            CASE is_COOLING_LEFT OF
                UPMRacing_14E_StateMachine_IN_COOLING_OFF_LEFT: 
                    (* During 'COOLING_OFF_LEFT': '<S1>:602' *)
                    (* '<S1>:603:1' sf_internal_predicateOutput = Cooling_Enable == true; *)

                    IF Cooling_Enable THEN 
                        (* Transition: '<S1>:603' *)
                        (* Exit 'COOLING_OFF_LEFT': '<S1>:602' *)
                        (* '<S1>:602:4' Cooling_Pumps_On = false; *)
                        Cooling_Pumps_On := FALSE;
                        is_COOLING_LEFT := UPMRacing_14E_StateMachine_IN_FAN_OFF;
                        (* Entry 'FAN_OFF': '<S1>:546' *)
                    END_IF;

                UPMRacing_14E_StateMachine_IN_FAN_OFF: 
                    (* During 'FAN_OFF': '<S1>:546' *)
                    (* '<S1>:548:1' sf_internal_predicateOutput = (AMK_TempMotor2 > Motor_Upper_Temp) || ... *)
                    (* '<S1>:548:2' (AMK_TempMotor4 > Motor_Upper_Temp); *)

                    IF (AMK_TempMotor2 > Motor_Upper_Temp) OR (AMK_TempMotor4 > Motor_Upper_Temp) THEN 
                        (* Transition: '<S1>:548' *)
                        is_COOLING_LEFT := UPMRacing_14E_StateMachine_IN_FAN_ON;
                        (* Entry 'FAN_ON': '<S1>:545' *)
                    ELSE 
                        (* '<S1>:604:1' sf_internal_predicateOutput = Cooling_Enable == false; *)

                        IF  NOT Cooling_Enable THEN 
                            (* Transition: '<S1>:604' *)
                            is_COOLING_LEFT := UPMRacing_14E_StateMachine_IN_COOLING_OFF_LEFT;
                            (* Entry 'COOLING_OFF_LEFT': '<S1>:602' *)
                            (* '<S1>:602:2' Cooling_Pumps_On = false; *)
                            Cooling_Pumps_On := FALSE;
                            (* '<S1>:602:3' Fan_Left = false; *)
                            Fan_Left := FALSE;
                        ELSE 
                            (* '<S1>:553:1' sf_internal_predicateOutput = (AMK_TempInverter1 > Inv_Upper_Temp) || ... *)
                            (* '<S1>:553:2' (AMK_TempInverter2 > Inv_Upper_Temp) || ... *)
                            (* '<S1>:553:3' (AMK_TempInverter3 > Inv_Upper_Temp) || ... *)
                            (* '<S1>:553:4' (AMK_TempInverter4 > Inv_Upper_Temp); *)

                            IF (((AMK_TempInverter1 > Inv_Upper_Temp) OR (AMK_TempInverter2 > Inv_Upper_Temp)) OR (AMK_TempInverter3 > Inv_Upper_Temp)) OR (AMK_TempInverter4 > Inv_Upper_Temp) THEN 
                                (* Transition: '<S1>:553' *)
                                is_COOLING_LEFT := UPMRacing_14E_StateMachine_IN_FAN_ON;
                                (* Entry 'FAN_ON': '<S1>:545' *)
                            ELSE 
                                (* '<S1>:546:2' Fan_Left = false; *)
                                Fan_Left := FALSE;
                            END_IF;

                        END_IF;

                    END_IF;

                UPMRacing_14E_StateMachine_IN_FAN_OFF_Speed: 
                    (* During 'FAN_OFF_Speed': '<S1>:544' *)
                    (* '<S1>:549:1' sf_internal_predicateOutput = Speed<Fan_Lower_Speed; *)

                    IF Speed < UINT_TO_REAL(Fan_Lower_Speed) THEN 
                        (* Transition: '<S1>:549' *)
                        is_COOLING_LEFT := UPMRacing_14E_StateMachine_IN_FAN_ON;
                        (* Entry 'FAN_ON': '<S1>:545' *)
                    ELSE 
                        (* '<S1>:606:1' sf_internal_predicateOutput = Cooling_Enable == false; *)

                        IF  NOT Cooling_Enable THEN 
                            (* Transition: '<S1>:606' *)
                            is_COOLING_LEFT := UPMRacing_14E_StateMachine_IN_COOLING_OFF_LEFT;
                            (* Entry 'COOLING_OFF_LEFT': '<S1>:602' *)
                            (* '<S1>:602:2' Cooling_Pumps_On = false; *)
                            Cooling_Pumps_On := FALSE;
                            (* '<S1>:602:3' Fan_Left = false; *)
                            Fan_Left := FALSE;
                        ELSE 
                            (* '<S1>:544:2' Fan_Left = false; *)
                            Fan_Left := FALSE;
                        END_IF;

                    END_IF;

                ELSE
                    (* During 'FAN_ON': '<S1>:545' *)
                    (* '<S1>:551:1' sf_internal_predicateOutput = (AMK_TempMotor2 < Motor_Lower_Temp) &amp; ... *)
                    (* '<S1>:551:2' (AMK_TempMotor4 < Motor_Lower_Temp) &amp; ... *)
                    (* '<S1>:551:3' (AMK_TempInverter1 < Inv_Lower_Temp) &amp; ... *)
                    (* '<S1>:551:4' (AMK_TempInverter2 < Inv_Lower_Temp) &amp; ... *)
                    (* '<S1>:551:5' (AMK_TempInverter3 < Inv_Lower_Temp) &amp; ... *)
                    (* '<S1>:551:6' (AMK_TempInverter4 < Inv_Lower_Temp); *)

                    IF (((((AMK_TempMotor2 < Motor_Lower_Temp) AND (AMK_TempMotor4 < Motor_Lower_Temp)) AND (AMK_TempInverter1 < Inv_Lower_Temp)) AND (AMK_TempInverter2 < Inv_Lower_Temp)) AND (AMK_TempInverter3 < Inv_Lower_Temp)) AND (AMK_TempInverter4 < Inv_Lower_Temp) THEN 
                        (* Transition: '<S1>:551' *)
                        is_COOLING_LEFT := UPMRacing_14E_StateMachine_IN_FAN_OFF;
                        (* Entry 'FAN_OFF': '<S1>:546' *)
                    ELSE 
                        (* '<S1>:605:1' sf_internal_predicateOutput = Cooling_Enable == false; *)

                        IF  NOT Cooling_Enable THEN 
                            (* Transition: '<S1>:605' *)
                            is_COOLING_LEFT := UPMRacing_14E_StateMachine_IN_COOLING_OFF_LEFT;
                            (* Entry 'COOLING_OFF_LEFT': '<S1>:602' *)
                            (* '<S1>:602:2' Cooling_Pumps_On = false; *)
                            Cooling_Pumps_On := FALSE;
                            (* '<S1>:602:3' Fan_Left = false; *)
                            Fan_Left := FALSE;
                        ELSE 
                            (* '<S1>:550:1' sf_internal_predicateOutput = Speed>Fan_Upper_Speed; *)

                            IF Speed > UINT_TO_REAL(Fan_Upper_Speed) THEN 
                                (* Transition: '<S1>:550' *)
                                is_COOLING_LEFT := UPMRacing_14E_StateMachine_IN_FAN_OFF_Speed;
                                (* Entry 'FAN_OFF_Speed': '<S1>:544' *)
                            ELSE 
                                (* '<S1>:545:2' Fan_Left = false; *)
                                Fan_Left := FALSE;
                            END_IF;

                        END_IF;

                    END_IF;

            END_CASE;

        END_IF;

        (* End of Chart: '<Root>/UPMRacing_14E_StateMachine' *)
END_CASE;

CAN_TX_V_1_4(
	
	
		(*AIM*)
		Estado_CAN:=Estado,
		Info_Inverter_Error_CAN:=Info_Inverter_Error,
		Estado_Error_CAN:=Estado_Error,
		Brake_Light_CAN:=Brake_Light,
		Pre_Charge_CAN:=Pre_Charge,
		Throttle_CAN := Throttle,
			
		AIM_TempMotor1_CAN:= AIM_TempMotor1,
		AIM_TempMotor2_CAN:= AIM_TempMotor2,
		AIM_TempMotor3_CAN:= AIM_TempMotor3,
		AIM_TempMotor4_CAN:= AIM_TempMotor4,
		
		AIM_TempInverter1_CAN := AIM_TempInverter1,
		AIM_TempInverter2_CAN := AIM_TempInverter2,
		AIM_TempInverter3_CAN := AIM_TempInverter3,		
		AIM_TempInverter4_CAN := AIM_TempInverter4,
		
		AIM_TempIGBT1_CAN := AIM_TempIGBT1,
		AIM_TempIGBT2_CAN := AIM_TempIGBT2,
		AIM_TempIGBT3_CAN := AIM_TempIGBT3,
		AIM_TempIGBT4_CAN := AIM_TempIGBT4,	
	
		AIM_bDerating1_CAN := AIM_bDerating1,
		AIM_bDerating2_CAN := AIM_bDerating2,
		AIM_bDerating3_CAN := AIM_bDerating3,
		AIM_bDerating4_CAN := AIM_bDerating4,
		
		K15_Value := DWORD_TO_WORD(GVL.K15),
		
		AIM_TorqueCurrent1_CAN := AIM_TorqueCurrent1,
		AIM_TorqueCurrent2_CAN := AIM_TorqueCurrent2,
		AIM_TorqueCurrent3_CAN := AIM_TorqueCurrent3,
		AIM_TorqueCurrent4_CAN := AIM_TorqueCurrent4,
		
		AIM_MagnetizingCurrent1_CAN := AIM_MagnetizingCurrent1, 
		AIM_MagnetizingCurrent2_CAN := AIM_MagnetizingCurrent2,
		AIM_MagnetizingCurrent3_CAN := AIM_MagnetizingCurrent3,
		AIM_MagnetizingCurrent4_CAN := AIM_MagnetizingCurrent4,
	
		AIM_TargetVelocity1_CAN := AIM_TargetVelocity1,
		AIM_TargetVelocity2_CAN := AIM_TargetVelocity2,
		AIM_TargetVelocity3_CAN := AIM_TargetVelocity3,
		AIM_TargetVelocity4_CAN := AIM_TargetVelocity4,
		
		AIM_TorqueLimitPositiv1_CAN := AIM_TorqueLimitPositiv1,
		AIM_TorqueLimitPositiv2_CAN := AIM_TorqueLimitPositiv2,
		AIM_TorqueLimitPositiv3_CAN := AIM_TorqueLimitPositiv3,
		AIM_TorqueLimitPositiv4_CAN := AIM_TorqueLimitPositiv4,
		
		AIM_ActualVelocity1_CAN := AIM_ActualVelocity1,
		AIM_ActualVelocity2_CAN := AIM_ActualVelocity2,
		AIM_ActualVelocity3_CAN := AIM_ActualVelocity3,
		AIM_ActualVelocity4_CAN := AIM_ActualVelocity4,
						
		Speed_RPM_CAN:= Speed_RPM,
		
		AIM_ErrorInfo1_CAN := AIM_ErrorInfo1,
		AIM_ErrorInfo2_CAN := AIM_ErrorInfo2,
		AIM_ErrorInfo3_CAN := AIM_ErrorInfo3,
		AIM_ErrorInfo4_CAN := AIM_ErrorInfo4,
		
		AIM_bError1_CAN := AIM_bError1,
		AIM_bError2_CAN := AIM_bError2,
		AIM_bError3_CAN := AIM_bError3,
		AIM_bError4_CAN := AIM_bError4
				
		(*FIN AIM*)
			);
(*__*)


CAN_TX_Inverters(
	
		(*INVERTERS*)
		AMK_bInverterOn1_CAN:=AMK_bInverterOn1,
		AMK_bDcOn1_CAN:=AMK_bDcOn1,
		AMK_bEnable1_CAN:=AMK_bEnable1,
		AMK_bErrorReset1_CAN:=AMK_bErrorReset1,
		AMK_TargetVelocity1_CAN:=AMK_TargetVelocity1,
		AMK_TorqueLimitPositiv1_CAN:=AMK_TorqueLimitPositiv1,
		AMK_TorqueLimitNegativ1_CAN:=AMK_TorqueLimitNegativ1,
		
		AMK_bInverterOn2_CAN:=AMK_bInverterOn2,
		AMK_bDcOn2_CAN:=AMK_bDcOn2,
		AMK_bEnable2_CAN:=AMK_bEnable2,
		AMK_bErrorReset2_CAN:=AMK_bErrorReset2,
		AMK_TargetVelocity2_CAN:=AMK_TargetVelocity2,
		AMK_TorqueLimitPositiv2_CAN:=AMK_TorqueLimitPositiv2,
		AMK_TorqueLimitNegativ2_CAN:=AMK_TorqueLimitNegativ2,
		
		AMK_bInverterOn3_CAN:=AMK_bInverterOn3,
		AMK_bDcOn3_CAN:=AMK_bDcOn3,
		AMK_bEnable3_CAN:=AMK_bEnable3,
		AMK_bErrorReset3_CAN:=AMK_bErrorReset3,
		AMK_TargetVelocity3_CAN:=AMK_TargetVelocity3,
		AMK_TorqueLimitPositiv3_CAN:=AMK_TorqueLimitPositiv3,
		AMK_TorqueLimitNegativ3_CAN:=AMK_TorqueLimitNegativ3,
		
		AMK_bInverterOn4_CAN:=AMK_bInverterOn4,
		AMK_bDcOn4_CAN:=AMK_bDcOn4,
		AMK_bEnable4_CAN:=AMK_bEnable4,
		AMK_bErrorReset4_CAN:=AMK_bErrorReset4,
		AMK_TargetVelocity4_CAN:=AMK_TargetVelocity4,
		AMK_TorqueLimitPositiv4_CAN:=AMK_TorqueLimitPositiv4,
		AMK_TorqueLimitNegativ4_CAN:=AMK_TorqueLimitNegativ4
		
		(*FIN INVERTERS*)
		
		);
		
(*__*)

END_FUNCTION_BLOCK

// Device/Application/CAN_Tx/CAN2_TX_V_0


FUNCTION_BLOCK CAN2_TX_V_0
VAR_INPUT
	
		//Cooling_Control
		Cooling_Pumps_Left_CAN: BOOL;
		Cooling_Pumps_Right_CAN: BOOL;
		Cooling_Pumps_INV_CAN: BOOL;		
		Fan_Left_CAN: BOOL;
		Fan_Right_CAN: BOOL;
		Fan_INV_CAN: BOOL;
		
		
END_VAR
VAR_OUTPUT
END_VAR
VAR
(*CanTX*) 

	(*Auxiliary Variable*)
		TxData: ARRAY [0..7]OF BYTE;
	
	(*Cooling_Control*)	
		Cooling_Control:CanTx;              (* Function block to send one CAN message *)
		
		

END_VAR

(*--------------------------------------------------Sensors TX-------------------------------------------------------------*)
(*Cooling_Control, ID=096h, 100 ms *) // State Variables
		(*TxData=16#00*)
			TxData[0]:=16#00;
			TxData[1]:=16#00;
			TxData[2]:=16#00;
			TxData[3]:=16#00;
			TxData[4]:=16#00;
			TxData[5]:=16#00;
			TxData[6]:=16#00;
			TxData[7]:=16#00;
		(*ASIGNACION DE LA VARIABLE A LA VARIABLE A ENVIAR (TxData)*)
		TxData[0].0:=Cooling_Pumps_Left_CAN;
		
		TxData[0].1:=Cooling_Pumps_Right_CAN;
		
		TxData[0].2:=Cooling_Pumps_INV_CAN;
		
		TxData[0].3:=Fan_Left_CAN;
		
		TxData[0].4:=Fan_Right_CAN;
		
		TxData[0].5:=Fan_INV_CAN;
		
		
									
				(*ENVÍO DE TxData*)
					Cooling_Control(	iEnable				:= TRUE, 			(* Enables sending of messages *)
									iCAN				:= ADR(GVL.H_CAN_TX_2),			(* Structure for sending / receiving CAN messages *)
									iForceSend			:= FALSE,                       (* Force sending sends message immediately *)
									iTransmitRate		:= T#100MS, 						(* Cyclic transmission every 100ms *)
									iCanId				:= 16#096,						(* CAN Id for message to send *)
									iCanIdExtended		:= FALSE, 						(* Standard CAN Frame *)
									iByteCount			:= 8,							(* Number of bytes to send *)
									iData				:= TxData, 						(* Data frame *)
									oTransmitterId		=> ,
									oTooManyTransmitters=> , 
									oMsgSent			=> 
								);
(*__*)


(*-----------------------------------------------FIN Sensors TX--------------------------------------------------------------*)

END_FUNCTION_BLOCK

// Device/Application/V_1/UPMRacing_14E_StateMachine_vieja
FUNCTION_BLOCK UPMRacing_14E_StateMachine_vieja
VAR_INPUT
	ssMethodType: SINT;
	MISSION_STATUS: USINT;
	SDC: BOOL;
	FRONT_AXLE_TRQ_REQUEST: UINT;
	REAR_AXLE_TRQ_REQUEST: UINT;
	STEER_REQUEST_deg: REAL;
	DIRECTION_REQUEST: BOOL;
	Accel_longitudinal_ms2: INT;
	Accel_lateral_ms2: INT;
	Yaw_rate_degps: INT;
	HANDSHAKE: BOOL;
	ESTOP_REQUEST: BOOL;
	LAP_COUNTER: USINT;
	CONES_COUNT_ACTUAL: USINT;
	CONES_COUNT_ALL: USINT;
	VEH_SPEED_ACTUAL: USINT;
	VEH_SPEED_DEMAND: USINT;
	FRONT_MOTOR_SPEED_MAX: UINT;
	REAR_MOTOR_SPEED_MAX: UINT;
	HYD_PRESS_F_REQ_pct: USINT;
	HYD_PRESS_R_REQ_pct: USINT;
END_VAR
VAR_OUTPUT
	State_ASSI: USINT;
	Steer_actual_deg: SINT;
	AI_ESTOP_REQUEST: BOOL;
	BMS_FAULT: BOOL;
	FR_WHEEL_SPEED: UINT;
	FL_WHEEL_SPEED: UINT;
	RR_WHEEL_SPEED: UINT;
	RL_WHEEL_SPEED: UINT;
	MISSION_STATUS_FAULT: BOOL;
	GO_SIGNAL: BOOL;
	AUTONOMOUS_BRAKING_FAULT: BOOL;
	BRAKE_PLAUSIBILITY_FAULT: BOOL;
	AI_COMMS_LOST_FAULT: BOOL;
	STATUS_EBS: USINT;
	TS_SWITCH_STATUS: BOOL;
	
			//FBTX_VCU2LOG_Dynamics1 
		Speed_actual_kmh: USINT;
		Speed_target_kmh: USINT;
		Steer_target_deg: SINT;
		Brake_actual_pct: USINT;
		Brake_target_pct: USINT;
		Drive_trq_actual_pct: SINT;
		Drive_trq_target_pct: SINT;
		
//FBTX_VCU2LOG_Status 		
		State_EBS: USINT; 
		AMI_STATE: USINT;
		State_steering: BOOL;
		State_service_brake: USINT;
		
				//FBTX_VCU2AI_Status
		SHUTDOWN_REQUEST: BOOL;
		STEERING_STATUS: BOOL;
		AS_STATE: USINT;
		FAULT_STATUS: BOOL;
		WARNING_STATUS: BOOL;
		WARN_BATT_TEMP_HIGH: BOOL;
		WARN_BATT_SOC_LOW: BOOL;
		HVIL_OPEN_FAULT: BOOL;
		HVIL_SHORT_FAULT: BOOL;
		EBS_FAULT: BOOL;
		OFFBOARD_CHARGER_FAULT: BOOL;
		AI_COMMS_LOST: BOOL;
		CHARGE_PROCEDURE_FAULT: BOOL;
		SHUTDOWN_CAUSE: USINT;
		
		//FBTX_VCU2AI_Drive_F
		FRONT_AXLE_TRQ: INT;
		FRONT_AXLE_TRQ_MAX: UINT;
		
		//FBTX_VCU2AI_Drive_R
		REAR_AXLE_TRQ: INT;
		REAR_AXLE_TRQ_MAX: UINT;
		
				//FBTX_VCU2AI_Steer
		ANGLE: INT;
		ANGLE_MAX: UINT;
		ANGLE_REQUEST: INT;
		
		//FBTX_VCU2AI_Brake 	
		HYD_PRESS_F_pct: USINT;
		HYD_PRESS_R_pct: USINT;
		STATUS_BRK: USINT;
		
		//FBTX_VCU2AI_Wheel_counts
		FL_PULSE_COUNT: UINT;
		FR_PULSE_COUNT: UINT;
		RL_PULSE_COUNT: UINT;
		RR_PULSE_COUNT: UINT;
		
		//VCU_STATUS
		SM_SYS: USINT;
		SM_AS: USINT;
		R1_AI2VCU_STATUS_TIMEOUT_ERROR: BOOL;
		R1_AI2VCU_DRIVE_F_TIMEOUT_ERROR: BOOL;
		R1_AI2VCU_DRIVE_R_TIMEOUT_ERROR: BOOL;
		R1_AI2VCU_STATUS_HANDSHAKE_ERROR: BOOL;
		R1_AI2VCU_STEER_TIMEOUT_ERROR: BOOL;
		R1_AI2VCU_BRAKE_TIMEOUT_ERROR: BOOL;
		SYS_ACTION_STATE: USINT;
		WARN_BRAKE_PLAUSIBILITY: BOOL;
		WARN_KL15_UNDER_V: BOOL;
		WARN_AI_ESTOP_REQ: BOOL;
		WARN_AI_COMMS_LOST: BOOL;
		WARN_AUTO_BRAKING: BOOL;
		WARN_MISSION_STATUS: BOOL;

		
		
END_VAR
VAR
	sf_internal_predicateOutput: BOOL;
	c_is_active_c3_UPMRacing_Dr: USINT;
	is_Main: USINT;
	temporalCounter_i1: PLC_CODER_TIMER;
	AS_SWITCH_STATUS: BOOL;
	//Llamadas a las funciones de CAN (Copiar)

	
//	CAN3_RX_V_0:CAN3_RX_V_0;	
	CAN2_RX_V_0:CAN2_RX_V_0;
	CAN1_RX_V_0:CAN1_RX_V_0;
	
	CAN2_TX_V_1:CAN2_TX_V_1;
	CAN1_TX_V_0:CAN1_TX_V_0;
	
END_VAR

CAN1_RX_V_0(
		
					Accel_longitudinal_ms2_CAN => Accel_longitudinal_ms2,
					Accel_lateral_ms2_CAN => Accel_lateral_ms2,
					Yaw_rate_degps_CAN => Yaw_rate_degps,
					HANDSHAKE_CAN => HANDSHAKE,
					ESTOP_REQUEST_CAN => ESTOP_REQUEST,
					MISSION_STATUS_CAN => MISSION_STATUS,
					DIRECTION_REQUEST_CAN => DIRECTION_REQUEST,
					LAP_COUNTER_CAN => LAP_COUNTER,
					CONES_COUNT_ACTUAL_CAN => CONES_COUNT_ACTUAL,
					CONES_COUNT_ALL_CAN => CONES_COUNT_ALL,
					VEH_SPEED_ACTUAL_CAN => VEH_SPEED_ACTUAL,
					VEH_SPEED_DEMAND_CAN => VEH_SPEED_DEMAND,
					FRONT_AXLE_TRQ_REQUEST_CAN => FRONT_AXLE_TRQ_REQUEST,
					FRONT_MOTOR_SPEED_MAX_CAN => FRONT_MOTOR_SPEED_MAX,
					REAR_AXLE_TRQ_REQUEST_CAN => REAR_AXLE_TRQ_REQUEST,
					REAR_MOTOR_SPEED_MAX_CAN => REAR_MOTOR_SPEED_MAX,
					STEER_REQUEST_deg_CAN => STEER_REQUEST_deg,
					HYD_PRESS_F_REQ_pct_CAN => HYD_PRESS_F_REQ_pct,
					HYD_PRESS_R_REQ_pct_CAN => HYD_PRESS_R_REQ_pct,

);
	(* *)
		 
CAN2_RX_V_0(
					ASMS_CAN => AS_SWITCH_STATUS,
					TSMS_CAN => TS_SWITCH_STATUS,
					GO_SIGNAL_CAN => GO_SIGNAL,
					SDC_CAN => SDC,
					MISSION_STATUS_FAULT_CAN => MISSION_STATUS_FAULT,
					AUTONOMOUS_BRAKING_FAULT_CAN => AUTONOMOUS_BRAKING_FAULT,
					COMMS_LOST_REQUEST_CAN => AI_COMMS_LOST_FAULT,
					BMS_FAULT_CAN => BMS_FAULT,
					EBS_Status_CAN => STATUS_EBS,
					FL_WHEEL_SPEED_CAN => FL_WHEEL_SPEED,
					FR_WHEEL_SPEED_CAN => FR_WHEEL_SPEED,
					RL_WHEEL_SPEED_CAN => RL_WHEEL_SPEED,
					RR_WHEEL_SPEED_CAN => RR_WHEEL_SPEED,
	
		);
	
	
CASE ssMethodType OF
    0: 
        (* SystemInitialize for Chart: '<Root>/UPMRacing_Driverless_V1 ' *)
        is_Main := 0;
        temporalCounter_i1(timerAction := 1, maxTime := 0);
        c_is_active_c3_UPMRacing_Dr := 0;
    1: 
        (* Chart: '<Root>/UPMRacing_Driverless_V1 ' incorporates:
         *  Inport: '<Root>/STEER_REQUEST_deg'
         *  Outport: '<Root>/AI_COMMS_LOST_FAULT'
         *  Outport: '<Root>/AI_ESTOP_REQUEST'
         *  Outport: '<Root>/AUTONOMOUS_BRAKING_FAULT'
         *  Outport: '<Root>/BMS_FAULT'
         *  Outport: '<Root>/BRAKE_PLAUSIBILITY_FAULT'
         *  Outport: '<Root>/FL_WHEEL_SPEED'
         *  Outport: '<Root>/FR_WHEEL_SPEED'
         *  Outport: '<Root>/GO_SIGNAL'
         *  Outport: '<Root>/MISSION_STATUS_FAULT'
         *  Outport: '<Root>/RL_WHEEL_SPEED'
         *  Outport: '<Root>/RR_WHEEL_SPEED'
         *  Outport: '<Root>/STATUS_EBS'
         *  Outport: '<Root>/Steer_actual_deg'
         *  Outport: '<Root>/TS_SWITCH_STATUS' *)
        (* Gateway: UPMRacing_Driverless_V1 *)
        (* During: UPMRacing_Driverless_V1 *)

        IF c_is_active_c3_UPMRacing_Dr = 0 THEN 
            (* Entry: UPMRacing_Driverless_V1 *)
            c_is_active_c3_UPMRacing_Dr := 1;
            (* Entry Internal: UPMRacing_Driverless_V1 *)
            (* Entry Internal 'Main': '<S1>:1349' *)
            (* Transition: '<S1>:1388' *)
            is_Main := 3;
            (* Outport: '<Root>/State_ASSI' *)
            (* Entry 'AS_OFF': '<S1>:1350' *)
            (* '<S1>:1350:3' State_ASSI = 1 *)
            State_ASSI := 1;
        ELSE 
            (* During 'Main': '<S1>:1349' *)

            CASE is_Main OF
                1: 
                    (* Outport: '<Root>/State_ASSI' *)
                    State_ASSI := 3;
                    (* During 'AS_DRIVING': '<S1>:1355' *)
                    (* '<S1>:1368:1' sf_internal_predicateOutput = MISSION_STATUS == 3 &amp;... *)
                    (* '<S1>:1368:2' FR_WHEEL_SPEED<10 &amp;... *)
                    (* '<S1>:1368:3' FL_WHEEL_SPEED<10 &amp;... *)
                    (* '<S1>:1368:4' RR_WHEEL_SPEED<10 &amp;... *)
                    (* '<S1>:1368:5' RL_WHEEL_SPEED<10; *)

                    IF ((((MISSION_STATUS = 3) AND (FR_WHEEL_SPEED < 10)) AND (FL_WHEEL_SPEED < 10)) AND (RR_WHEEL_SPEED < 10)) AND (RL_WHEEL_SPEED < 10) THEN 
                        (* Transition: '<S1>:1368' *)
                        is_Main := 2;
                        (* Outport: '<Root>/State_ASSI' *)
                        (* Entry 'AS_FINISHED': '<S1>:1354' *)
                        (* '<S1>:1354:3' State_ASSI=5 *)
                        State_ASSI := 5;
                    ELSE 
                        (* '<S1>:1373:1' sf_internal_predicateOutput = SDC==0 ||... *)
                        (* '<S1>:1373:2' AS_SWITCH_STATUS == 0 ||... *)
                        (* '<S1>:1373:3' GO_SIGNAL == 0 ||... *)
                        (* '<S1>:1373:4' MISSION_STATUS_FAULT == 1 ||... *)
                        (* '<S1>:1373:5' AUTONOMOUS_BRAKING_FAULT == 1 || ...  *)
                        (* '<S1>:1373:6' BRAKE_PLAUSIBILITY_FAULT == 1 ||... *)
                        (* '<S1>:1373:7' AI_ESTOP_REQUEST == 1 ||... *)
                        (* '<S1>:1373:8' AI_COMMS_LOST_FAULT == 1 ||... *)
                        (* '<S1>:1373:9' BMS_FAULT == 1 ||... *)
                        (* '<S1>:1373:10' STATUS_EBS == 1; *)

                        IF ((((((((( NOT SDC) OR ( NOT AS_SWITCH_STATUS)) OR ( NOT GO_SIGNAL)) OR MISSION_STATUS_FAULT) OR AUTONOMOUS_BRAKING_FAULT) OR BRAKE_PLAUSIBILITY_FAULT) OR AI_ESTOP_REQUEST) OR AI_COMMS_LOST_FAULT) OR BMS_FAULT) OR (STATUS_EBS = 1) THEN 
                            (* Transition: '<S1>:1373' *)
                            is_Main := 5;
                            temporalCounter_i1(timerAction := 1, maxTime := 0);
                            (* Outport: '<Root>/State_ASSI' *)
                            (* Entry 'EMERGENCY_BRAKE': '<S1>:1353' *)
                            (* '<S1>:1353:3' State_ASSI=4 *)
                            State_ASSI := 4;
                        END_IF;

                    END_IF;

                2: 
                    (* Outport: '<Root>/State_ASSI' *)
                    State_ASSI := 5;
                    (* During 'AS_FINISHED': '<S1>:1354' *)
                    (* '<S1>:1366:1' sf_internal_predicateOutput = AS_SWITCH_STATUS == 0; *)

                    IF  NOT AS_SWITCH_STATUS THEN 
                        (* Transition: '<S1>:1366' *)
                        is_Main := 3;
                        (* Outport: '<Root>/State_ASSI' *)
                        (* Entry 'AS_OFF': '<S1>:1350' *)
                        (* '<S1>:1350:3' State_ASSI = 1 *)
                        State_ASSI := 1;
                    ELSE 
                        (* '<S1>:1367:1' sf_internal_predicateOutput = SDC==0; *)

                        IF  NOT SDC THEN 
                            (* Transition: '<S1>:1367' *)
                            is_Main := 5;
                            temporalCounter_i1(timerAction := 1, maxTime := 0);
                            (* Outport: '<Root>/State_ASSI' *)
                            (* Entry 'EMERGENCY_BRAKE': '<S1>:1353' *)
                            (* '<S1>:1353:3' State_ASSI=4 *)
                            State_ASSI := 4;
                        END_IF;

                    END_IF;

                3: 
                    (* Outport: '<Root>/State_ASSI' *)
                    State_ASSI := 1;
                    (* During 'AS_OFF': '<S1>:1350' *)
                    (* '<S1>:1356:1' sf_internal_predicateOutput = AS_SWITCH_STATUS == 1 &amp;... *)
                    (* '<S1>:1356:2' TS_SWITCH_STATUS == 1 &amp;... *)
                    (* '<S1>:1356:3' STATUS_EBS == 2 &amp;... *)
                    (* '<S1>:1356:4' MISSION_STATUS == 1; *)

                    IF ((AS_SWITCH_STATUS AND TS_SWITCH_STATUS) AND (STATUS_EBS = 2)) AND (MISSION_STATUS = 1) THEN 
                        (* Transition: '<S1>:1356' *)
                        is_Main := 4;
                        temporalCounter_i1(timerAction := 1, maxTime := 0);
                        (* Outport: '<Root>/State_ASSI' *)
                        (* Entry 'AS_READY': '<S1>:1352' *)
                        (* '<S1>:1352:3' State_ASSI=2 *)
                        State_ASSI := 2;
                    END_IF;

                4: 
                    (* Outport: '<Root>/State_ASSI' *)
                    State_ASSI := 2;
                    (* During 'AS_READY': '<S1>:1352' *)
                    (* '<S1>:1358:1' sf_internal_predicateOutput = AS_SWITCH_STATUS == 0; *)

                    IF  NOT AS_SWITCH_STATUS THEN 
                        (* Transition: '<S1>:1358' *)
                        is_Main := 3;
                        (* Outport: '<Root>/State_ASSI' *)
                        (* Entry 'AS_OFF': '<S1>:1350' *)
                        (* '<S1>:1350:3' State_ASSI = 1 *)
                        State_ASSI := 1;
                    ELSE 
                        (* '<S1>:1374:1' sf_internal_predicateOutput = SDC==0; *)

                        IF  NOT SDC THEN 
                            (* Transition: '<S1>:1374' *)
                            is_Main := 5;
                            temporalCounter_i1(timerAction := 1, maxTime := 0);
                            (* Outport: '<Root>/State_ASSI' *)
                            (* Entry 'EMERGENCY_BRAKE': '<S1>:1353' *)
                            (* '<S1>:1353:3' State_ASSI=4 *)
                            State_ASSI := 4;
                        ELSE 
                            (* '<S1>:1413:1' sf_internal_predicateOutput = after(5,sec) &amp;... *)
                            (* '<S1>:1413:2' FRONT_AXLE_TRQ_REQUEST == 0 &amp;... *)
                            (* '<S1>:1413:3' REAR_AXLE_TRQ_REQUEST  == 0 &amp;... *)
                            (* '<S1>:1413:4' STEER_REQUEST_deg  == 0 &amp;... *)
                            (* '<S1>:1413:5' Steer_actual_deg < 5  &amp;... *)
                            (* '<S1>:1413:6' DIRECTION_REQUEST == 0 &amp;... *)
                            (* '<S1>:1413:7' GO_SIGNAL == 0; *)
                            temporalCounter_i1(timerAction := 2, maxTime := 5000);
                            sf_internal_predicateOutput := temporalCounter_i1.done;

                            IF (((((sf_internal_predicateOutput AND (FRONT_AXLE_TRQ_REQUEST = 0)) AND (REAR_AXLE_TRQ_REQUEST = 0)) AND (STEER_REQUEST_deg = 0)) AND (Steer_actual_deg < 5)) AND ( NOT DIRECTION_REQUEST)) AND ( NOT GO_SIGNAL) THEN 
                                (* Transition: '<S1>:1413' *)
                                is_Main := 7;
                                (* Entry 'INTERMIDIATE': '<S1>:1412' *)
                                (* '<S1>:1412:3' State_ASSI=2 *)
                            END_IF;

                        END_IF;

                    END_IF;

                5: 
                    (* Outport: '<Root>/State_ASSI' *)
                    State_ASSI := 4;
                    (* During 'EMERGENCY_BRAKE': '<S1>:1353' *)
                    (* '<S1>:1363:1' sf_internal_predicateOutput = after(15,sec); *)
                    temporalCounter_i1(timerAction := 2, maxTime := 15000);

                    IF temporalCounter_i1.done THEN 
                        (* Transition: '<S1>:1363' *)
                        is_Main := 6;
                        (* Entry 'EMERGENCY_BRAKE_COMPLETED': '<S1>:1414' *)
                        (* '<S1>:1414:3' State_ASSI=4 *)
                    END_IF;

                6: 
                    (* Outport: '<Root>/State_ASSI' *)
                    State_ASSI := 4;
                    (* During 'EMERGENCY_BRAKE_COMPLETED': '<S1>:1414' *)
                    (* '<S1>:1416:1' sf_internal_predicateOutput = AS_SWITCH_STATUS == 0; *)

                    IF  NOT AS_SWITCH_STATUS THEN 
                        (* Transition: '<S1>:1416' *)
                        is_Main := 3;
                        (* Outport: '<Root>/State_ASSI' *)
                        (* Entry 'AS_OFF': '<S1>:1350' *)
                        (* '<S1>:1350:3' State_ASSI = 1 *)
                        State_ASSI := 1;
                    END_IF;

                ELSE
                    (* Outport: '<Root>/State_ASSI' *)
                    State_ASSI := 2;
                    (* During 'INTERMIDIATE': '<S1>:1412' *)
                    (* '<S1>:1372:1' sf_internal_predicateOutput = GO_SIGNAL == 1; *)

                    IF GO_SIGNAL THEN 
                        (* Transition: '<S1>:1372' *)
                        is_Main := 1;
                        (* Outport: '<Root>/State_ASSI' *)
                        (* Entry 'AS_DRIVING': '<S1>:1355' *)
                        (* '<S1>:1355:3' State_ASSI=3 *)
                        State_ASSI := 3;
                    END_IF;

            END_CASE;

        END_IF;
		AS_STATE := State_ASSI;

        (* End of Chart: '<Root>/UPMRacing_Driverless_V1 ' *)
END_CASE;


CAN1_TX_V_0(
				//FBTX_VCU2LOG_Dynamics1 
		Speed_actual_kmh_CAN := Speed_actual_kmh,
		Speed_target_kmh_CAN := Speed_target_kmh,
		Steer_actual_deg_CAN := Steer_actual_deg,
		Steer_target_deg_CAN := Steer_target_deg,
		Brake_actual_pct_CAN := Brake_actual_pct, 
		Brake_target_pct_CAN := Brake_target_pct, 
		Drive_trq_actual_pct_CAN := Drive_trq_actual_pct,
		Drive_trq_target_pct_CAN := Drive_trq_target_pct, 
		
	
		//FBTX_VCU2LOG_Status 		
		State_ASSI_CAN := State_ASSI,
		State_EBS_CAN := State_EBS,  
//		AMI_STATE_CAN := AMI_STATE, 
		State_steering_CAN := State_steering, 
		State_service_brake_CAN := State_service_brake,
		
		//FBTX_VCU2AI_Status
		HANDSHAKE_CAN := HANDSHAKE,
		SHUTDOWN_REQUEST_CAN := SHUTDOWN_REQUEST,
		AS_SWITCH_STATUS_CAN := AS_SWITCH_STATUS ,
		TS_SWITCH_STATUS_CAN := TS_SWITCH_STATUS,
		GO_SIGNAL_CAN := GO_SIGNAL,
		STEERING_STATUS_CAN := STEERING_STATUS,
		AS_STATE_CAN := AS_STATE,
		FAULT_STATUS_CAN := FAULT_STATUS,
		WARNING_STATUS_CAN := WARNING_STATUS,
		WARN_BATT_TEMP_HIGH_CAN := WARN_BATT_TEMP_HIGH,
		WARN_BATT_SOC_LOW_CAN := WARN_BATT_SOC_LOW,
		AI_ESTOP_REQUEST_CAN := AI_ESTOP_REQUEST,
		HVIL_OPEN_FAULT_CAN := HVIL_OPEN_FAULT,
		HVIL_SHORT_FAULT_CAN := HVIL_SHORT_FAULT, 
		EBS_FAULT_CAN := EBS_FAULT,
		OFFBOARD_CHARGER_FAULT_CAN := OFFBOARD_CHARGER_FAULT,
		AI_COMMS_LOST_CAN := AI_COMMS_LOST,
		AUTONOMOUS_BRAKING_FAULT_CAN := AUTONOMOUS_BRAKING_FAULT,
		MISSION_STATUS_FAULT_CAN := MISSION_STATUS_FAULT, 
		CHARGE_PROCEDURE_FAULT_CAN := CHARGE_PROCEDURE_FAULT,
		BMS_FAULT_CAN := BMS_FAULT, 
		BRAKE_PLAUSIBILITY_FAULT_CAN := BRAKE_PLAUSIBILITY_FAULT, 
		SHUTDOWN_CAUSE_CAN := SHUTDOWN_CAUSE,
		
		//FBTX_VCU2AI_Drive_F
		FRONT_AXLE_TRQ_CAN := FRONT_AXLE_TRQ, 
		FRONT_AXLE_TRQ_REQUEST_CAN := FRONT_AXLE_TRQ_REQUEST,
		FRONT_AXLE_TRQ_MAX_CAN := FRONT_AXLE_TRQ_MAX, 
		
		//FBTX_VCU2AI_Drive_R
		REAR_AXLE_TRQ_CAN := REAR_AXLE_TRQ,
		REAR_AXLE_TRQ_REQUEST_CAN := REAR_AXLE_TRQ_REQUEST,
		REAR_AXLE_TRQ_MAX_CAN := REAR_AXLE_TRQ_MAX,
		
		//FBTX_VCU2AI_Steer
		ANGLE_CAN := ANGLE,
		ANGLE_MAX_CAN := ANGLE_MAX,
		ANGLE_REQUEST_CAN := ANGLE_REQUEST,
		
		//FBTX_VCU2AI_Brake 	
		HYD_PRESS_F_pct_CAN := HYD_PRESS_F_pct, 
		HYD_PRESS_F_REQ_pct_CAN := HYD_PRESS_F_REQ_pct,
		HYD_PRESS_R_pct_CAN := HYD_PRESS_R_pct,
		HYD_PRESS_R_REQ_pct_CAN := HYD_PRESS_R_REQ_pct,
		STATUS_BRK_CAN := STATUS_BRK,
		STATUS_EBS_CAN := STATUS_EBS, 
		
		//FBTX_VCU2AI_Speeds
		FL_WHEEL_SPEED_CAN := FL_WHEEL_SPEED,
    	FR_WHEEL_SPEED_CAN := FR_WHEEL_SPEED, 
	    RL_WHEEL_SPEED_CAN := RL_WHEEL_SPEED,
    	RR_WHEEL_SPEED_CAN := RR_WHEEL_SPEED, 
		
		//FBTX_VCU2AI_Wheel_counts
		FL_PULSE_COUNT_CAN := FL_PULSE_COUNT,
		FR_PULSE_COUNT_CAN := FR_PULSE_COUNT, 
		RL_PULSE_COUNT_CAN := RL_PULSE_COUNT,
		RR_PULSE_COUNT_CAN := RR_PULSE_COUNT,
		
		//VCU_STATUS
		SM_SYS_CAN := SM_SYS, 
		SM_AS_CAN := SM_AS,
		R1_AI2VCU_STATUS_TIMEOUT_ERROR_CAN := R1_AI2VCU_STATUS_TIMEOUT_ERROR,
		R1_AI2VCU_DRIVE_F_TIMEOUT_ERROR_CAN := R1_AI2VCU_DRIVE_F_TIMEOUT_ERROR,
		R1_AI2VCU_DRIVE_R_TIMEOUT_ERROR_CAN := R1_AI2VCU_DRIVE_R_TIMEOUT_ERROR, 
		R1_AI2VCU_STATUS_HANDSHAKE_ERROR_CAN := R1_AI2VCU_STATUS_HANDSHAKE_ERROR,
		R1_AI2VCU_STEER_TIMEOUT_ERROR_CAN := R1_AI2VCU_STEER_TIMEOUT_ERROR, 
		R1_AI2VCU_BRAKE_TIMEOUT_ERROR_CAN := R1_AI2VCU_BRAKE_TIMEOUT_ERROR,
		SYS_ACTION_STATE_CAN := SYS_ACTION_STATE,
		WARN_BRAKE_PLAUSIBILITY_CAN := WARN_BRAKE_PLAUSIBILITY, 
		WARN_KL15_UNDER_V_CAN := WARN_KL15_UNDER_V,
		WARN_AI_ESTOP_REQ_CAN := WARN_AI_ESTOP_REQ,
		WARN_AI_COMMS_LOST_CAN := WARN_AI_COMMS_LOST,
		WARN_AUTO_BRAKING_CAN := WARN_AUTO_BRAKING,
		WARN_MISSION_STATUS_CAN := WARN_MISSION_STATUS,
		

);
 


(*__*)

END_FUNCTION_BLOCK
